// TIA Portal project "Project" (V17)

(* hardware
DEVICE "S71500/ET200MP station_1"  S7-1500 station
   slot 0: "Rail_0"  Rack  6ES7 590-1***0-0AA0
   slot 1: "PLC_1"  CPU 1511-1 PN  6ES7 511-1AK00-0AB0  V1.8
      slot 3: "CPU display_1"  6ES7591-1AA00-0AA0
DEVICE "PC-System_1"  SIMATIC PC station
   slot 0: "SIMATIC PC station"  Rail  SIMATIC PC-Station  V1.0
      slot 125: "Stationmanager"  Station_Manager  V6.0.4
   slot 1: "HMI_RT_1"  WinCC RT Professional  6AV2 105-0xxxx-xxxx  17.0.0.0
   slot 2: "IE general_1"  IE General  IE_CP  V8.2.0
      slot 1: "PROFINET interface"  IEGeneral.Interface.8.2.0
*)

// ===== PLC "PLC_1"  CPU 1511-1 PN =====

VAR_GLOBAL   // PLC tag table "Default tag table"
   "Brake_Out" AT %M0.0 : Bool;
   "Baffle_Out" AT %MW18 : Int;
   "RPM_In" AT %MW2 : Int;
   "OilTemp_In" AT %MW4 : Int;
   "Baffle_En" AT %M0.1 : Bool;
   "Current_In" AT %MW6 : Int;
   "OilPumpVFDsp_Out" AT %MW8 : Int;
   "OilPumpVFDen_Out" AT %M0.2 : Bool;
   "OilFlow_In" AT %MW10 : Int;
   "ProgLang" AT %MW12 : Int;
   "ONS1" AT %M0.3 : Bool;
   "PB_LAD" AT %M0.4 : Bool;
   "PB_FBD" AT %M0.5 : Bool;
   "PB_SCL" AT %M0.6 : Bool;
   "PB_STL" AT %M0.7 : Bool;
   "ONS" AT %M1.0 : Bool;
   "ONS2" AT %M1.1 : Bool;
   "ONS3" AT %M1.2 : Bool;
   "AlarmHorn_Out" AT %M1.3 : Bool;
   "StationInterlock_Out" AT %M1.4 : Bool;
   "OilPumpVFDpct" AT %MW14 : Int;
   "Bafflepct" AT %MW16 : Int;
   "OilTemp" AT %MW20 : Int;
   "OilFlow" AT %MW22 : Int;
   "RPM" AT %MW24 : Int;
   "Current" AT %MW26 : Int;
   "OilPumpVFDOff_PB" AT %M1.5 : Bool;
   "OilPumpVFDHand_PB" AT %M1.6 : Bool;
   "OilPumpVFDAuto_PB" AT %M1.7 : Bool;
   "OilPumpVFDHoa" AT %MW28 : Int;
   "BrakeOff_PB" AT %M2.0 : Bool;
   "BrakeHand_PB" AT %M2.1 : Bool;
   "BrakeAuto_PB" AT %M2.2 : Bool;
   "BrakeHoa" AT %MW30 : Int;
   "AlarmHornOff_PB" AT %M2.3 : Bool;
   "AlarmHornHand_PB" AT %M2.4 : Bool;
   "AlarmHornAuto_PB" AT %M2.5 : Bool;
   "AlarmHornHoa" AT %MW32 : Int;
   "StationInterlockOff_PB" AT %M2.6 : Bool;
   "StationInterlockHand_PB" AT %M2.7 : Bool;
   "StationInterlockAuto_PB" AT %M3.0 : Bool;
   "StationInterlockHoa" AT %MW34 : Int;
   "OilPumpVFD_Ctrl" AT %M3.1 : Bool;
   "Brake_Ctrl" AT %M3.2 : Bool;
   "AlarmHorn_Ctrl" AT %M3.3 : Bool;
   "StationInterlock_Ctrl" AT %M3.4 : Bool;
END_VAR

DATA_BLOCK "SimLogic_DB"   // DB1
{ S7_Optimized_Access := 'TRUE' }
VERSION : 0.1
// stored: InstanceOfName SimLogic
"SimLogic"
BEGIN
END_DATA_BLOCK

DATA_BLOCK "IO_LAD_DB"   // DB2
{ S7_Optimized_Access := 'TRUE' }
VERSION : 0.1
// stored: InstanceOfName IO_LAD
"IO_LAD"
BEGIN
END_DATA_BLOCK

DATA_BLOCK "IO_STL_DB"   // DB4
{ S7_Optimized_Access := 'TRUE' }
VERSION : 0.1
// stored: InstanceOfName IO_STL
"IO_STL"
BEGIN
END_DATA_BLOCK

DATA_BLOCK "IO_SCL_DB"   // DB5
{ S7_Optimized_Access := 'TRUE' }
VERSION : 0.1
// stored: InstanceOfName IO_SCL
"IO_SCL"
BEGIN
END_DATA_BLOCK

DATA_BLOCK "IO_FBD_DB"   // DB6
{ S7_Optimized_Access := 'TRUE' }
VERSION : 0.1
// stored: InstanceOfName IO_FBD
"IO_FBD"
BEGIN
END_DATA_BLOCK

DATA_BLOCK "ALARMS_LAD_DB"   // DB7
{ S7_Optimized_Access := 'TRUE' }
VERSION : 0.1
// stored: InstanceOfName ALARMS_LAD
"ALARMS_LAD"
BEGIN
END_DATA_BLOCK

DATA_BLOCK "HOA_LAD_DB"   // DB8
{ S7_Optimized_Access := 'TRUE' }
VERSION : 0.1
// stored: InstanceOfName HOA_LAD
"HOA_LAD"
BEGIN
END_DATA_BLOCK

DATA_BLOCK "HOA_FBD_DB"   // DB9
{ S7_Optimized_Access := 'TRUE' }
VERSION : 0.1
// stored: InstanceOfName HOA_FBD
"HOA_FBD"
BEGIN
END_DATA_BLOCK

DATA_BLOCK "HOA_SCL_DB"   // DB10
{ S7_Optimized_Access := 'TRUE' }
VERSION : 0.1
// stored: InstanceOfName HOA_SCL
"HOA_SCL"
BEGIN
END_DATA_BLOCK

DATA_BLOCK "HOA_STL_DB"   // DB11
{ S7_Optimized_Access := 'TRUE' }
VERSION : 0.1
// stored: InstanceOfName HOA_STL
"HOA_STL"
BEGIN
END_DATA_BLOCK

// folder: System blocks/Program resources

DATA_BLOCK "IEC_Timer_0_DB_25"   // DB3
{ S7_Optimized_Access := 'TRUE' }
AUTHOR : Simatic
FAMILY : IEC
NAME : IEC_TMR
VERSION : 1.0
// stored: InstanceOfName IEC_TIMER
"IEC_TIMER"
BEGIN
END_DATA_BLOCK

DATA_BLOCK "IEC_Timer_0_DB"   // DB17
{ S7_Optimized_Access := 'TRUE' }
AUTHOR : Simatic
FAMILY : IEC
NAME : IEC_TMR
VERSION : 1.0
// stored: InstanceOfName IEC_TIMER
"IEC_TIMER"
BEGIN
END_DATA_BLOCK

DATA_BLOCK "IEC_Timer_1_DB"   // DB43
{ S7_Optimized_Access := 'TRUE' }
AUTHOR : Simatic
FAMILY : IEC
NAME : IEC_TMR
VERSION : 1.0
// stored: InstanceOfName IEC_TIMER
"IEC_TIMER"
BEGIN
END_DATA_BLOCK

// folder: (top level)

FUNCTION_BLOCK "SimLogic"   // FB1, FBD
{ S7_Optimized_Access := 'TRUE' }
VERSION : 0.1
   VAR
      "TO" : Bool;
      rpmv : Int;
      addrpmv : Bool;
      otsp : Int;
      ott : Int;
      TO1 : Bool;
      TO2 : Bool;
      be2 : Int;
      be3 : Int;
      be1 : Int;
      TO3 : Bool;
   END_VAR
   VAR_TEMP
      bf : Int;
      rpmvt : Int;
      bfr : Real;
   END_VAR
BEGIN

REGION Network 1
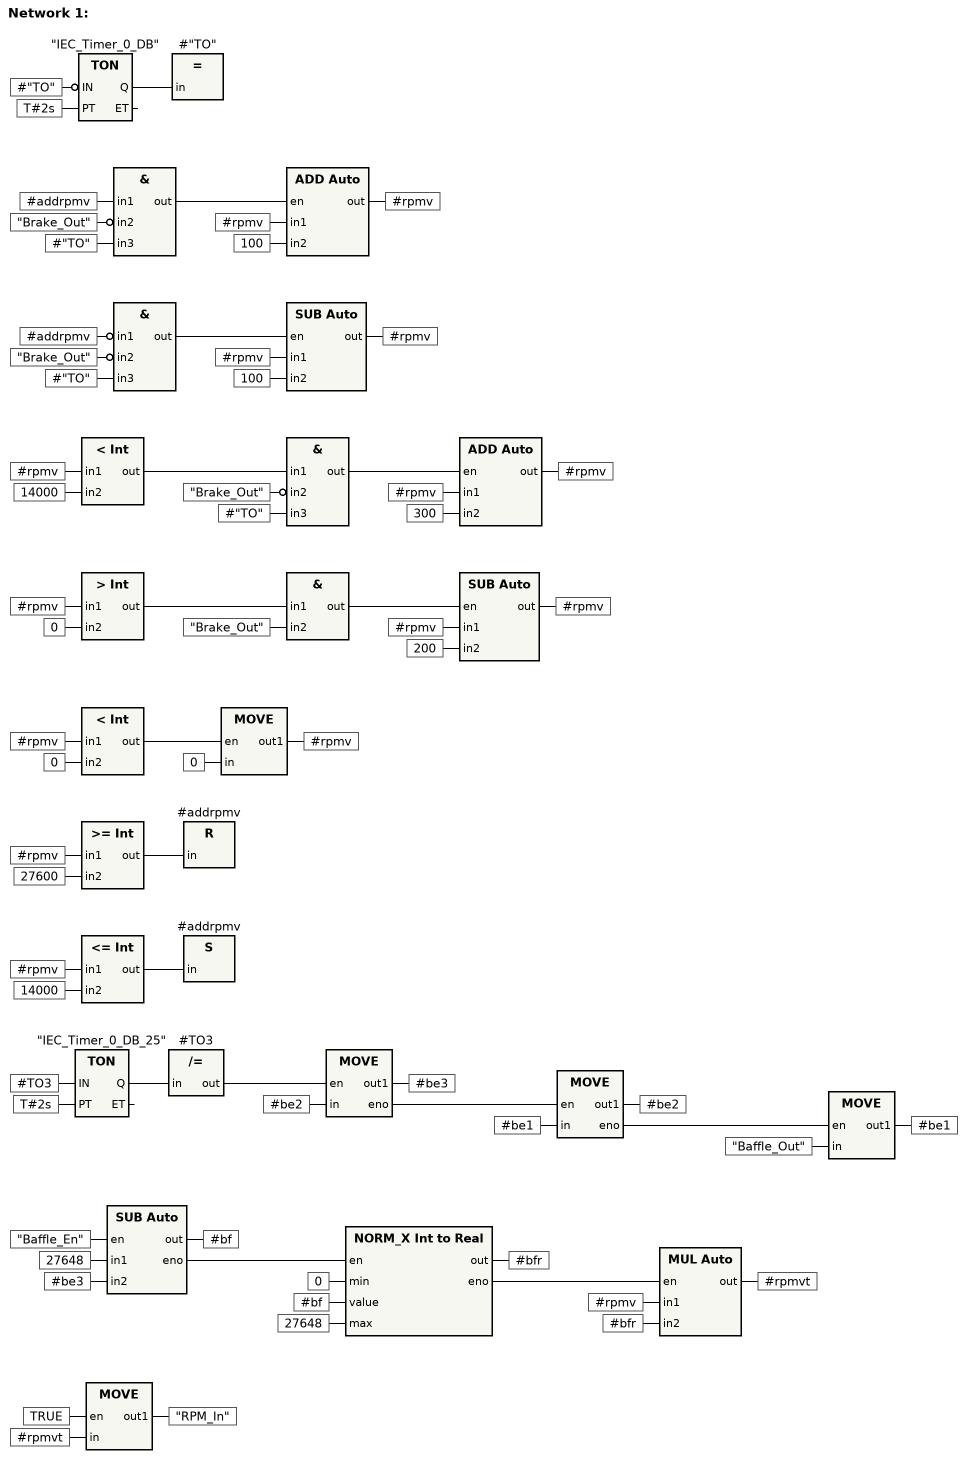
   "IEC_Timer_0_DB".TON(IN := NOT #"TO", PT := T#2s);
   #"TO" := "IEC_Timer_0_DB".Q;
   IF #addrpmv AND NOT "Brake_Out" AND #"TO" THEN #rpmv := #rpmv + 100; END_IF;
   IF NOT #addrpmv AND NOT "Brake_Out" AND #"TO" THEN #rpmv := #rpmv - 100; END_IF;
   IF (#rpmv < 14000) AND NOT "Brake_Out" AND #"TO" THEN #rpmv := #rpmv + 300; END_IF;
   IF (#rpmv > 0) AND "Brake_Out" THEN #rpmv := #rpmv - 200; END_IF;
   IF #rpmv < 0 THEN #rpmv := 0; END_IF;
   IF #rpmv >= 27600 THEN #addrpmv := FALSE; END_IF;
   IF #rpmv <= 14000 THEN #addrpmv := TRUE; END_IF;
   "IEC_Timer_0_DB_25".TON(IN := #TO3, PT := T#2s);
   #TO3 := NOT "IEC_Timer_0_DB_25".Q;
   IF "IEC_Timer_0_DB_25".Q THEN
       #be3 := #be2;
       #be2 := #be1;
       #be1 := "Baffle_Out";
   END_IF;
   IF "Baffle_En" THEN
       #bf := 27648 - #be3;
       #bfr := NORM_X(MIN := 0, VALUE := #bf, MAX := 27648);
       #rpmvt := #rpmv * #bfr;
   END_IF;
   IF TRUE THEN "RPM_In" := #rpmvt; END_IF;
END_REGION

REGION Network 2
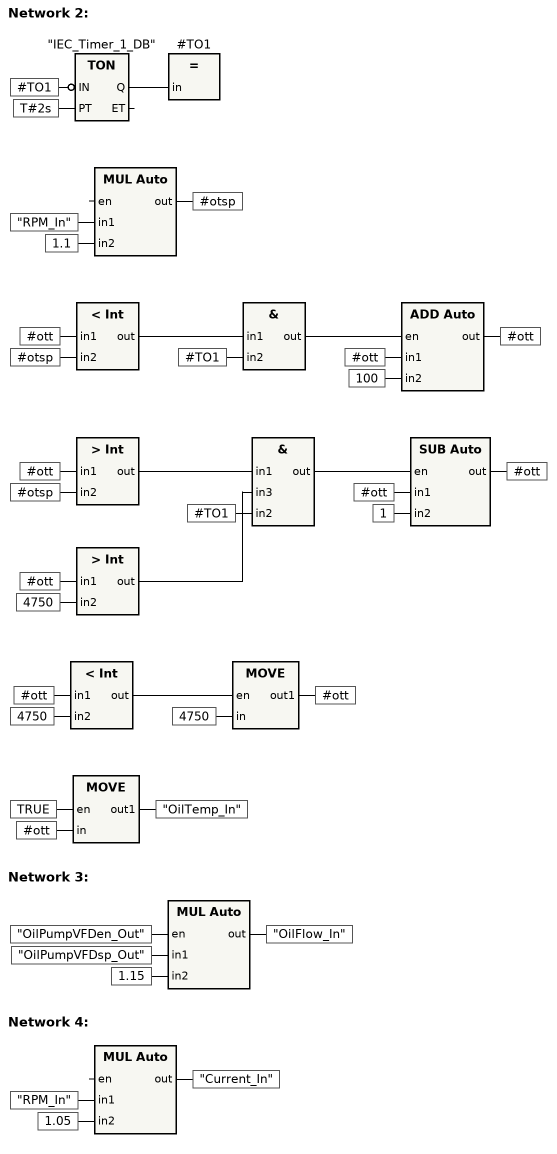
   "IEC_Timer_1_DB".TON(IN := NOT #TO1, PT := T#2s);
   #TO1 := "IEC_Timer_1_DB".Q;
   #otsp := "RPM_In" * 1.1;
   IF (#ott < #otsp) AND #TO1 THEN #ott := #ott + 100; END_IF;
   IF (#ott > #otsp) AND (#ott > 4750) AND #TO1 THEN #ott := #ott - 1; END_IF;
   IF #ott < 4750 THEN #ott := 4750; END_IF;
   IF TRUE THEN "OilTemp_In" := #ott; END_IF;
END_REGION

REGION Network 3
   IF "OilPumpVFDen_Out" THEN "OilFlow_In" := "OilPumpVFDsp_Out" * 1.15; END_IF;
END_REGION

REGION Network 4
   "Current_In" := "RPM_In" * 1.05;
END_REGION
END_FUNCTION_BLOCK

FUNCTION_BLOCK "IO_LAD"   // FB2, LAD
{ S7_Optimized_Access := 'TRUE' }
VERSION : 0.1
BEGIN

REGION Network 1: Digital Outputs
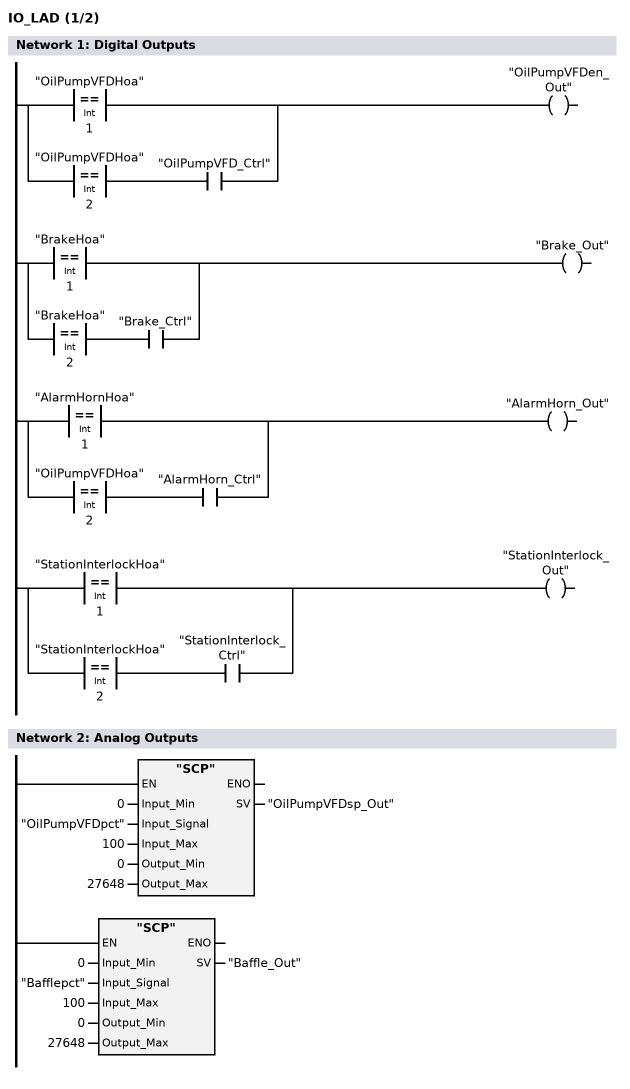
   RUNG wire#powerrail
      { S7_Templates := "SrcType := Int" } EQ_Contact(in1 := "OilPumpVFDHoa", in2 := 1)
      wire#w1
      Coil( "OilPumpVFDen_Out" )
   END_RUNG
   RUNG wire#powerrail
      { S7_Templates := "SrcType := Int" } EQ_Contact(in1 := "OilPumpVFDHoa", in2 := 2)
      Contact( "OilPumpVFD_Ctrl" )
   END_RUNG wire#w1
   RUNG wire#powerrail
      { S7_Templates := "SrcType := Int" } EQ_Contact(in1 := "BrakeHoa", in2 := 1)
      wire#w2
      Coil( "Brake_Out" )
   END_RUNG
   RUNG wire#powerrail
      { S7_Templates := "SrcType := Int" } EQ_Contact(in1 := "BrakeHoa", in2 := 2)
      Contact( "Brake_Ctrl" )
   END_RUNG wire#w2
   RUNG wire#powerrail
      { S7_Templates := "SrcType := Int" } EQ_Contact(in1 := "AlarmHornHoa", in2 := 1)
      wire#w3
      Coil( "AlarmHorn_Out" )
   END_RUNG
   RUNG wire#powerrail
      { S7_Templates := "SrcType := Int" } EQ_Contact(in1 := "OilPumpVFDHoa", in2 := 2)
      Contact( "AlarmHorn_Ctrl" )
   END_RUNG wire#w3
   RUNG wire#powerrail
      { S7_Templates := "SrcType := Int" } EQ_Contact(in1 := "StationInterlockHoa", in2 := 1)
      wire#w4
      Coil( "StationInterlock_Out" )
   END_RUNG
   RUNG wire#powerrail
      { S7_Templates := "SrcType := Int" } EQ_Contact(in1 := "StationInterlockHoa", in2 := 2)
      Contact( "StationInterlock_Ctrl" )
   END_RUNG wire#w4
   // the same network as SCL:
   "OilPumpVFDen_Out" := ("OilPumpVFDHoa" = 1) OR (("OilPumpVFDHoa" = 2) AND "OilPumpVFD_Ctrl");
   "Brake_Out" := ("BrakeHoa" = 1) OR (("BrakeHoa" = 2) AND "Brake_Ctrl");
   "AlarmHorn_Out" := ("AlarmHornHoa" = 1) OR (("OilPumpVFDHoa" = 2) AND "AlarmHorn_Ctrl");
   "StationInterlock_Out" := ("StationInterlockHoa" = 1) OR (("StationInterlockHoa" = 2) AND "StationInterlock_Ctrl");
END_REGION

REGION Network 2: Analog Outputs
   RUNG wire#powerrail
      "SCP"(Input_Min := 0, Input_Signal := "OilPumpVFDpct", Input_Max := 100, Output_Min := 0, Output_Max := 27648, SV => "OilPumpVFDsp_Out")
   END_RUNG
   RUNG wire#powerrail
      "SCP"(Input_Min := 0, Input_Signal := "Bafflepct", Input_Max := 100, Output_Min := 0, Output_Max := 27648, SV => "Baffle_Out")
   END_RUNG
   // the same network as SCL:
   "SCP"(Input_Min := 0,
         Input_Signal := "OilPumpVFDpct",
         Input_Max := 100,
         Output_Min := 0,
         Output_Max := 27648,
         SV => "OilPumpVFDsp_Out");
   "SCP"(Input_Min := 0,
         Input_Signal := "Bafflepct",
         Input_Max := 100,
         Output_Min := 0,
         Output_Max := 27648,
         SV => "Baffle_Out");
END_REGION

REGION Network 3: Analog Inputs
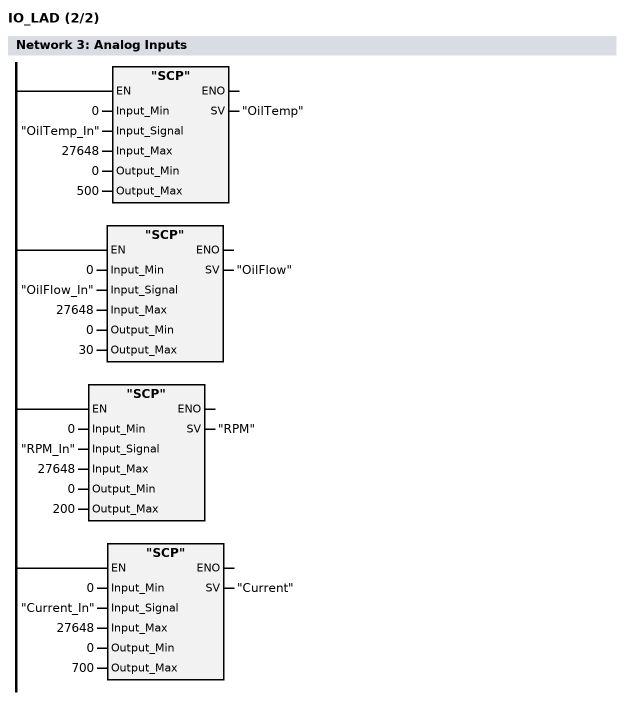
   RUNG wire#powerrail
      "SCP"(Input_Min := 0, Input_Signal := "OilTemp_In", Input_Max := 27648, Output_Min := 0, Output_Max := 500, SV => "OilTemp")
   END_RUNG
   RUNG wire#powerrail
      "SCP"(Input_Min := 0, Input_Signal := "OilFlow_In", Input_Max := 27648, Output_Min := 0, Output_Max := 30, SV => "OilFlow")
   END_RUNG
   RUNG wire#powerrail
      "SCP"(Input_Min := 0, Input_Signal := "RPM_In", Input_Max := 27648, Output_Min := 0, Output_Max := 200, SV => "RPM")
   END_RUNG
   RUNG wire#powerrail
      "SCP"(Input_Min := 0, Input_Signal := "Current_In", Input_Max := 27648, Output_Min := 0, Output_Max := 700, SV => "Current")
   END_RUNG
   // the same network as SCL:
   "SCP"(Input_Min := 0,
         Input_Signal := "OilTemp_In",
         Input_Max := 27648,
         Output_Min := 0,
         Output_Max := 500,
         SV => "OilTemp");
   "SCP"(Input_Min := 0,
         Input_Signal := "OilFlow_In",
         Input_Max := 27648,
         Output_Min := 0,
         Output_Max := 30,
         SV => "OilFlow");
   "SCP"(Input_Min := 0,
         Input_Signal := "RPM_In",
         Input_Max := 27648,
         Output_Min := 0,
         Output_Max := 200,
         SV => "RPM");
   "SCP"(Input_Min := 0,
         Input_Signal := "Current_In",
         Input_Max := 27648,
         Output_Min := 0,
         Output_Max := 700,
         SV => "Current");
END_REGION
END_FUNCTION_BLOCK

FUNCTION_BLOCK "IO_FBD"   // FB3, FBD
{ S7_Optimized_Access := 'TRUE' }
VERSION : 0.1
BEGIN

REGION Network 1: Digital Outputs
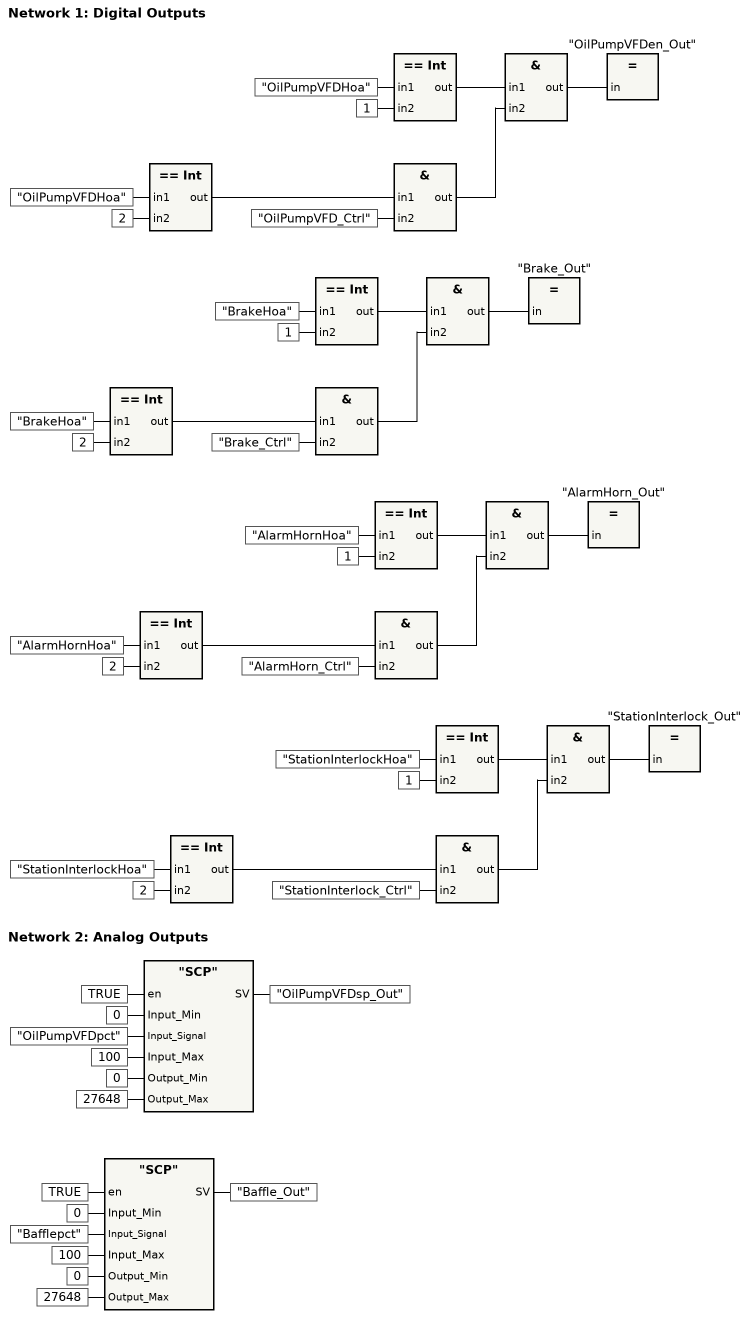
   "OilPumpVFDen_Out" := ("OilPumpVFDHoa" = 1) AND ("OilPumpVFDHoa" = 2) AND "OilPumpVFD_Ctrl";
   "Brake_Out" := ("BrakeHoa" = 1) AND ("BrakeHoa" = 2) AND "Brake_Ctrl";
   "AlarmHorn_Out" := ("AlarmHornHoa" = 1) AND ("AlarmHornHoa" = 2) AND "AlarmHorn_Ctrl";
   "StationInterlock_Out" := ("StationInterlockHoa" = 1) AND ("StationInterlockHoa" = 2) AND "StationInterlock_Ctrl";
END_REGION

REGION Network 2: Analog Outputs
   IF TRUE THEN
       "SCP"(Input_Min := 0,
             Input_Signal := "OilPumpVFDpct",
             Input_Max := 100,
             Output_Min := 0,
             Output_Max := 27648,
             SV => "OilPumpVFDsp_Out");
       "SCP"(Input_Min := 0,
             Input_Signal := "Bafflepct",
             Input_Max := 100,
             Output_Min := 0,
             Output_Max := 27648,
             SV => "Baffle_Out");
   END_IF;
END_REGION

REGION Network 3: Analog Inputs
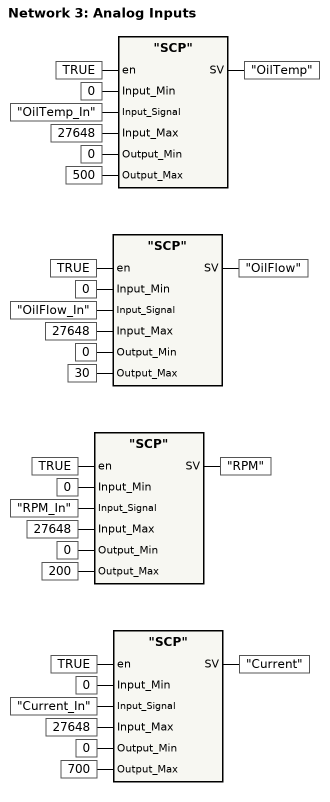
   IF TRUE THEN
       "SCP"(Input_Min := 0,
             Input_Signal := "OilTemp_In",
             Input_Max := 27648,
             Output_Min := 0,
             Output_Max := 500,
             SV => "OilTemp");
       "SCP"(Input_Min := 0,
             Input_Signal := "OilFlow_In",
             Input_Max := 27648,
             Output_Min := 0,
             Output_Max := 30,
             SV => "OilFlow");
       "SCP"(Input_Min := 0,
             Input_Signal := "RPM_In",
             Input_Max := 27648,
             Output_Min := 0,
             Output_Max := 200,
             SV => "RPM");
       "SCP"(Input_Min := 0,
             Input_Signal := "Current_In",
             Input_Max := 27648,
             Output_Min := 0,
             Output_Max := 700,
             SV => "Current");
   END_IF;
END_REGION
END_FUNCTION_BLOCK

FUNCTION_BLOCK "IO_SCL"   // FB4, SCL
{ S7_Optimized_Access := 'TRUE' }
VERSION : 0.1
BEGIN
   //Digital Ouputs
   IF "OilPumpVFDHoa" = 0 OR ("OilPumpVFDHoa" = 2 AND NOT "OilPumpVFD_Ctrl") THEN
       "OilPumpVFDen_Out" := 0;
   END_IF;

   IF "OilPumpVFDHoa" = 1 OR ("OilPumpVFDHoa" = 2 AND "OilPumpVFD_Ctrl") THEN
       "OilPumpVFDen_Out" := 1;
   END_IF;


   IF "BrakeHoa" = 0 OR ("BrakeHoa" = 2 AND NOT "Brake_Ctrl") THEN
       "Brake_Out" := 0;
   END_IF;

   IF "BrakeHoa" = 1 OR ("BrakeHoa" = 2 AND "Brake_Ctrl") THEN
       "Brake_Out" := 1;
   END_IF;


   IF "AlarmHornHoa" = 0 OR ("AlarmHornHoa" = 2 AND NOT "AlarmHorn_Ctrl") THEN
       "AlarmHorn_Out" := 0;
   END_IF;

   IF "AlarmHornHoa" = 1 OR ("AlarmHornHoa" = 2 AND "AlarmHorn_Ctrl") THEN
       "AlarmHorn_Out" := 1;
   END_IF;


   IF "StationInterlockHoa" = 0 OR ("StationInterlockHoa" = 2 AND NOT "StationInterlock_Ctrl") THEN
       "StationInterlock_Out" := 0;
   END_IF;

   IF "StationInterlockHoa" = 1 OR ("StationInterlockHoa" = 2 AND "StationInterlock_Ctrl") THEN
       "StationInterlock_Out" := 1;
   END_IF;

   // Analog Outputs
   "SCP"(Input_Min:=0,
         Input_Signal:="OilPumpVFDpct",
         Input_Max:=100,
         Output_Min:=0,
         Output_Max:=27648,
         SV=>"OilPumpVFDsp_Out");

   "SCP"(Input_Min := 0,
         Input_Signal := "Bafflepct",
         Input_Max := 100,
         Output_Min := 0,
         Output_Max := 27648,
         SV => "Baffle_Out");

   //Analog Inputs
   "SCP"(Input_Min := 0,
         Input_Signal := "OilTemp_In",
         Input_Max := 27648,
         Output_Min := 0,
         Output_Max := 500,
         SV => "OilTemp");

   "SCP"(Input_Min := 0,
         Input_Signal := "OilFlow_In",
         Input_Max := 27648,
         Output_Min := 0,
         Output_Max := 30,
         SV => "OilFlow");

   "SCP"(Input_Min := 0,
         Input_Signal := "RPM_In",
         Input_Max := 27648,
         Output_Min := 0,
         Output_Max := 200,
         SV => "RPM");

   "SCP"(Input_Min := 0,
         Input_Signal := "Current_In",
         Input_Max := 27648,
         Output_Min := 0,
         Output_Max := 700,
         SV => "Current");
END_FUNCTION_BLOCK

FUNCTION_BLOCK "IO_STL"   // FB5, STL
{ S7_Optimized_Access := 'TRUE' }
VERSION : 0.1
BEGIN

REGION Network 1
   //Digital Ouputs
   OilPumpVFD:L     "OilPumpVFDHoa";
         L     0;
         ==I;
         JC    ResetOilPumpVFD;
         CLR;
         L     "OilPumpVFDHoa";
         L     1;
         ==I;
         JC    SetOilPumpVFD;
         CLR;
         L     "OilPumpVFDHoa";
         L     2;
         ==I;
         JC    AutoOilPumpVFD;

   AutoOilPumpVFD:A     "OilPumpVFD_Ctrl";
         JC    SetOilPumpVFD;
         JU    Brake;
   SetOilPumpVFD:S     "OilPumpVFDen_Out";
         JU    Brake;
   ResetOilPumpVFD:R     "OilPumpVFDen_Out";
         JU    Brake;


   Brake:L     "BrakeHoa";
         L     0;
         ==I;
         JC    ResetBrake;
         CLR;
         L     "BrakeHoa";
         L     1;
         ==I;
         JC    SetBrake;
         CLR;
         L     "BrakeHoa";
         L     2;
         ==I;
         JC    AutoBrake;

   AutoBrake:A     "Brake_Ctrl";
         JC    SetBrake;
         JU    AlarmHorn;
   SetBrake:S     "Brake_Out";
         JU    AlarmHorn;
   ResetBrake:R     "Brake_Out";
         JU    AlarmHorn;

   AlarmHorn:L     "AlarmHornHoa";
         L     0;
         ==I;
         JC    ResetAlarmHorn;
         CLR;
         L     "AlarmHornHoa";
         L     1;
         ==I;
         JC    SetAlarmHorn;
         CLR;
         L     "AlarmHornHoa";
         L     2;
         ==I;
         JC    AutoAlarmHorn;

   AutoAlarmHorn:A     "AlarmHorn_Ctrl";
         JC    SetAlarmHorn;
         JU    StationInterlock;
   SetAlarmHorn:S     "AlarmHorn_Out";
         JU    StationInterlock;
   ResetAlarmHorn:R     "AlarmHorn_Out";
         JU    StationInterlock;

   StationInterlock:L     "StationInterlockHoa";
         L     0;
         ==I;
         JC    ResetStationInterlock;
         CLR;
         L     "StationInterlockHoa";
         L     1;
         ==I;
         JC    SetStationInterlock;
         CLR;
         L     "StationInterlockHoa";
         L     2;
         ==I;
         JC    AutoStationInterlock;

   AutoStationInterlock:A     "StationInterlock_Ctrl";
         JC    SetStationInterlock;
         JU    AnalogOutputs;
   SetStationInterlock:S     "StationInterlock_Out";
         JU    AnalogOutputs;
   ResetStationInterlock:R     "StationInterlock_Out";
         JU    AnalogOutputs;


   //Analog Outputs
   AnalogOutputs:CALL  "SCP"
         ( Input_Min    := 0,
           Input_Signal := "OilPumpVFDpct",
           Input_Max    := 100,
           Output_Min   := 0,
           Output_Max   := 27648,
           SV           := "OilPumpVFDsp_Out"
         );

         CALL  "SCP"
         ( Input_Min    := 0,
           Input_Signal := "Bafflepct",
           Input_Max    := 100,
           Output_Min   := 0,
           Output_Max   := 27648,
           SV           := "Baffle_Out"
         );

   //Analog Inputs
   AnalogInputs:CALL  "SCP"
         ( Input_Min    := 0,
           Input_Signal := "OilTemp_In",
           Input_Max    := 27648,
           Output_Min   := 0,
           Output_Max   := 500,
           SV           := "OilTemp"
         );

         CALL  "SCP"
         ( Input_Min    := 0,
           Input_Signal := "OilFlow_In",
           Input_Max    := 27648,
           Output_Min   := 0,
           Output_Max   := 30,
           SV           := "OilFlow"
         );

         CALL  "SCP"
         ( Input_Min    := 0,
           Input_Signal := "RPM_In",
           Input_Max    := 27648,
           Output_Min   := 0,
           Output_Max   := 200,
           SV           := "RPM"
         );

         CALL  "SCP"
         ( Input_Min    := 0,
           Input_Signal := "Current_In",
           Input_Max    := 27648,
           Output_Min   := 0,
           Output_Max   := 700,
           SV           := "Current"
         );
END_REGION
END_FUNCTION_BLOCK

FUNCTION_BLOCK "ALARMS_LAD"   // FB6, LAD
{ S7_Optimized_Access := 'TRUE' }
VERSION : 0.1
BEGIN
END_FUNCTION_BLOCK

FUNCTION_BLOCK "HOA_LAD"   // FB7, LAD
{ S7_Optimized_Access := 'TRUE' }
VERSION : 0.1
   VAR
      OS1 : Bool;
      OS2 : Bool;
      OS3 : Bool;
      OS4 : Bool;
      OS5 : Bool;
      OS6 : Bool;
      OS7 : Bool;
      OS8 : Bool;
      OS9 : Bool;
      OS10 : Bool;
      OS11 : Bool;
      OS12 : Bool;
   END_VAR
   VAR_TEMP   // added for the SCL form of the ladder/FBD networks
      _w1 : Bool;
      _w2 : Bool;
      _w3 : Bool;
   END_VAR
BEGIN

REGION Network 1: OilPumpVFD
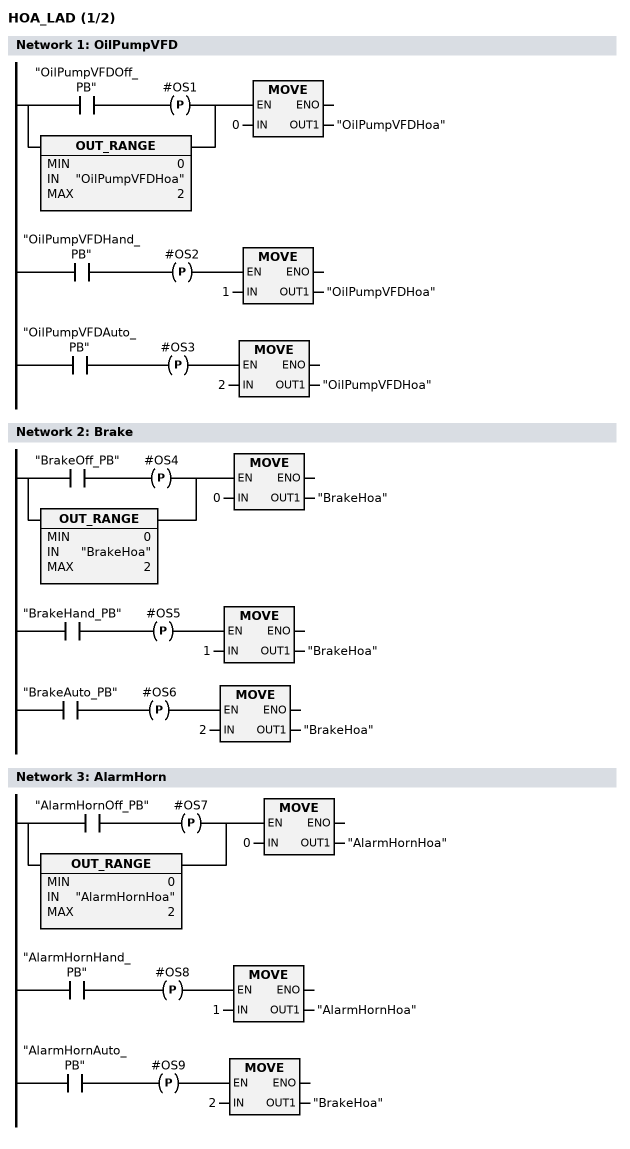
   #_w1 := "OilPumpVFDOff_PB" AND NOT #OS1;   // rising edge
   #OS1 := "OilPumpVFDOff_PB";
   IF #_w1 OR ("OilPumpVFDHoa" < 0) OR ("OilPumpVFDHoa" > 2) THEN "OilPumpVFDHoa" := 0; END_IF;
   #_w2 := "OilPumpVFDHand_PB" AND NOT #OS2;   // rising edge
   #OS2 := "OilPumpVFDHand_PB";
   IF #_w2 THEN "OilPumpVFDHoa" := 1; END_IF;
   #_w3 := "OilPumpVFDAuto_PB" AND NOT #OS3;   // rising edge
   #OS3 := "OilPumpVFDAuto_PB";
   IF #_w3 THEN "OilPumpVFDHoa" := 2; END_IF;
END_REGION

REGION Network 2: Brake
   #_w1 := "BrakeOff_PB" AND NOT #OS4;   // rising edge
   #OS4 := "BrakeOff_PB";
   IF #_w1 OR ("BrakeHoa" < 0) OR ("BrakeHoa" > 2) THEN "BrakeHoa" := 0; END_IF;
   #_w2 := "BrakeHand_PB" AND NOT #OS5;   // rising edge
   #OS5 := "BrakeHand_PB";
   IF #_w2 THEN "BrakeHoa" := 1; END_IF;
   #_w3 := "BrakeAuto_PB" AND NOT #OS6;   // rising edge
   #OS6 := "BrakeAuto_PB";
   IF #_w3 THEN "BrakeHoa" := 2; END_IF;
END_REGION

REGION Network 3: AlarmHorn
   #_w1 := "AlarmHornOff_PB" AND NOT #OS7;   // rising edge
   #OS7 := "AlarmHornOff_PB";
   IF #_w1 OR ("AlarmHornHoa" < 0) OR ("AlarmHornHoa" > 2) THEN "AlarmHornHoa" := 0; END_IF;
   #_w2 := "AlarmHornHand_PB" AND NOT #OS8;   // rising edge
   #OS8 := "AlarmHornHand_PB";
   IF #_w2 THEN "AlarmHornHoa" := 1; END_IF;
   #_w3 := "AlarmHornAuto_PB" AND NOT #OS9;   // rising edge
   #OS9 := "AlarmHornAuto_PB";
   IF #_w3 THEN "BrakeHoa" := 2; END_IF;
END_REGION

REGION Network 4: StationInterlock
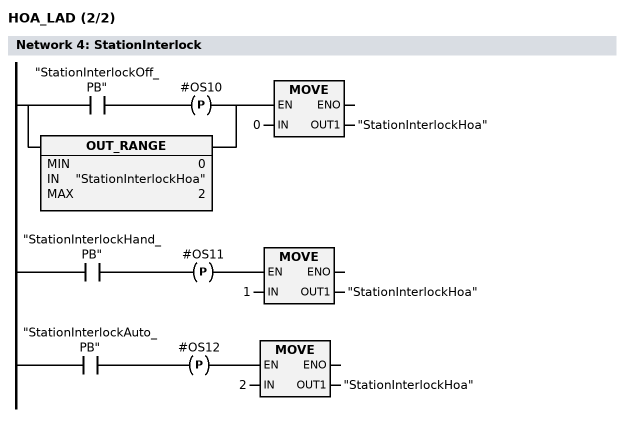
   #_w1 := "StationInterlockOff_PB" AND NOT #OS10;   // rising edge
   #OS10 := "StationInterlockOff_PB";
   IF #_w1 OR ("StationInterlockHoa" < 0) OR ("StationInterlockHoa" > 2) THEN
       "StationInterlockHoa" := 0;
   END_IF;
   #_w2 := "StationInterlockHand_PB" AND NOT #OS11;   // rising edge
   #OS11 := "StationInterlockHand_PB";
   IF #_w2 THEN "StationInterlockHoa" := 1; END_IF;
   #_w3 := "StationInterlockAuto_PB" AND NOT #OS12;   // rising edge
   #OS12 := "StationInterlockAuto_PB";
   IF #_w3 THEN "StationInterlockHoa" := 2; END_IF;
END_REGION
END_FUNCTION_BLOCK

FUNCTION_BLOCK "HOA_FBD"   // FB8, FBD
{ S7_Optimized_Access := 'TRUE' }
VERSION : 0.1
   VAR
      OS1 : Bool;
      OS2 : Bool;
      OS3 : Bool;
      OS4 : Bool;
      OS5 : Bool;
      OS6 : Bool;
      OS7 : Bool;
      OS8 : Bool;
      OS9 : Bool;
      OS10 : Bool;
      OS11 : Bool;
      OS12 : Bool;
   END_VAR
   VAR_TEMP   // added for the SCL form of the ladder/FBD networks
      _w1 : Bool;
      _w2 : Bool;
      _w3 : Bool;
   END_VAR
BEGIN

REGION Network 1: OilPumpVFD
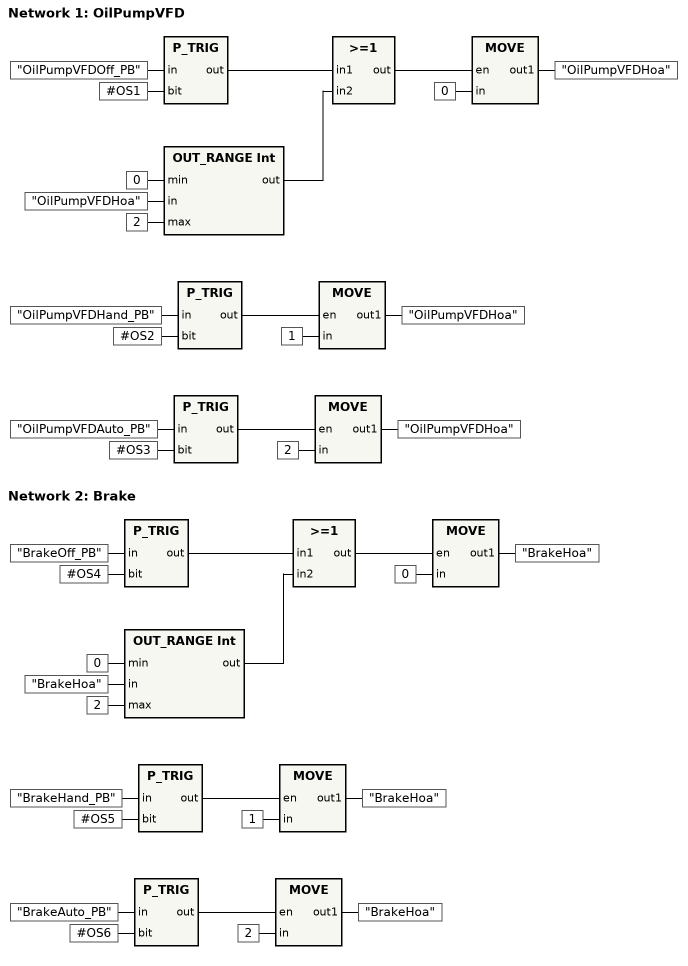
   #_w1 := "OilPumpVFDOff_PB" AND NOT #OS1;   // rising edge
   #OS1 := "OilPumpVFDOff_PB";
   IF #_w1 OR ("OilPumpVFDHoa" < 0) OR ("OilPumpVFDHoa" > 2) THEN "OilPumpVFDHoa" := 0; END_IF;
   #_w2 := "OilPumpVFDHand_PB" AND NOT #OS2;   // rising edge
   #OS2 := "OilPumpVFDHand_PB";
   IF #_w2 THEN "OilPumpVFDHoa" := 1; END_IF;
   #_w3 := "OilPumpVFDAuto_PB" AND NOT #OS3;   // rising edge
   #OS3 := "OilPumpVFDAuto_PB";
   IF #_w3 THEN "OilPumpVFDHoa" := 2; END_IF;
END_REGION

REGION Network 2: Brake
   #_w1 := "BrakeOff_PB" AND NOT #OS4;   // rising edge
   #OS4 := "BrakeOff_PB";
   IF #_w1 OR ("BrakeHoa" < 0) OR ("BrakeHoa" > 2) THEN "BrakeHoa" := 0; END_IF;
   #_w2 := "BrakeHand_PB" AND NOT #OS5;   // rising edge
   #OS5 := "BrakeHand_PB";
   IF #_w2 THEN "BrakeHoa" := 1; END_IF;
   #_w3 := "BrakeAuto_PB" AND NOT #OS6;   // rising edge
   #OS6 := "BrakeAuto_PB";
   IF #_w3 THEN "BrakeHoa" := 2; END_IF;
END_REGION

REGION Network 3: AlarmHorn
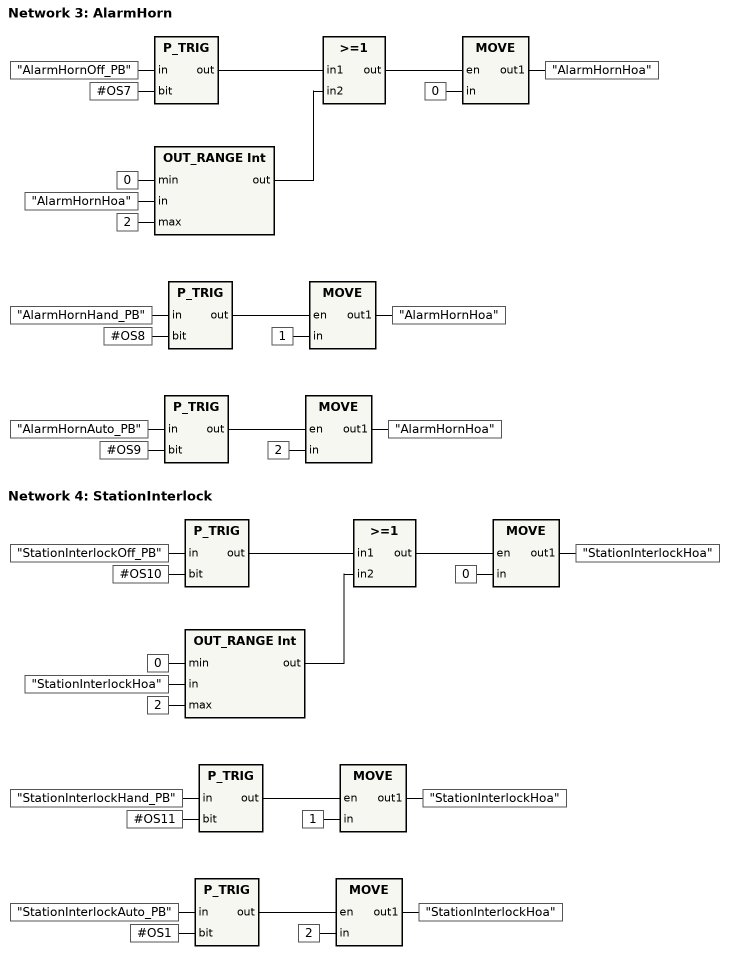
   #_w1 := "AlarmHornOff_PB" AND NOT #OS7;   // rising edge
   #OS7 := "AlarmHornOff_PB";
   IF #_w1 OR ("AlarmHornHoa" < 0) OR ("AlarmHornHoa" > 2) THEN "AlarmHornHoa" := 0; END_IF;
   #_w2 := "AlarmHornHand_PB" AND NOT #OS8;   // rising edge
   #OS8 := "AlarmHornHand_PB";
   IF #_w2 THEN "AlarmHornHoa" := 1; END_IF;
   #_w3 := "AlarmHornAuto_PB" AND NOT #OS9;   // rising edge
   #OS9 := "AlarmHornAuto_PB";
   IF #_w3 THEN "AlarmHornHoa" := 2; END_IF;
END_REGION

REGION Network 4: StationInterlock
   #_w1 := "StationInterlockOff_PB" AND NOT #OS10;   // rising edge
   #OS10 := "StationInterlockOff_PB";
   IF #_w1 OR ("StationInterlockHoa" < 0) OR ("StationInterlockHoa" > 2) THEN
       "StationInterlockHoa" := 0;
   END_IF;
   #_w2 := "StationInterlockHand_PB" AND NOT #OS11;   // rising edge
   #OS11 := "StationInterlockHand_PB";
   IF #_w2 THEN "StationInterlockHoa" := 1; END_IF;
   #_w3 := "StationInterlockAuto_PB" AND NOT #OS1;   // rising edge
   #OS1 := "StationInterlockAuto_PB";
   IF #_w3 THEN "StationInterlockHoa" := 2; END_IF;
END_REGION
END_FUNCTION_BLOCK

FUNCTION_BLOCK "HOA_SCL"   // FB9, SCL
{ S7_Optimized_Access := 'TRUE' }
VERSION : 0.1
BEGIN
   // OilPumpVFD
   IF "OilPumpVFDHoa" < 0 OR "OilPumpVFDHoa" > 2 THEN
       "OilPumpVFDHoa" := 0;
   END_IF;

   IF "OilPumpVFDOff_PB" AND "OilPumpVFDHoa" <> 0 THEN
       "OilPumpVFDHoa" := 0;
   END_IF;

   IF "OilPumpVFDHand_PB" AND "OilPumpVFDHoa" <> 1 THEN
       "OilPumpVFDHoa" := 1;
   END_IF;

   IF "OilPumpVFDAuto_PB" AND "OilPumpVFDHoa" <> 2 THEN
       "OilPumpVFDHoa" := 2;
   END_IF;

   //Brake
   IF "BrakeHoa" < 0 OR "BrakeHoa" > 2 THEN
       "BrakeHoa" := 0;
   END_IF;

   IF "BrakeOff_PB" AND "BrakeHoa" <> 0 THEN
       "BrakeHoa" := 0;
   END_IF;

   IF "BrakeHand_PB" AND "BrakeHoa" <> 1 THEN
       "BrakeHoa" := 1;
   END_IF;

   IF "BrakeAuto_PB" AND "BrakeHoa" <> 2 THEN
       "BrakeHoa" := 2;
   END_IF;

   //AlarmHorn
   IF "AlarmHornHoa" < 0 OR "AlarmHornHoa" > 2 THEN
       "AlarmHornHoa" := 0;
   END_IF;

   IF "AlarmHornOff_PB" AND "AlarmHornHoa" <> 0 THEN
       "AlarmHornHoa" := 0;
   END_IF;

   IF "AlarmHornHand_PB" AND "AlarmHornHoa" <> 1 THEN
       "AlarmHornHoa" := 1;
   END_IF;

   IF "AlarmHornAuto_PB" AND "AlarmHornHoa" <> 2 THEN
       "AlarmHornHoa" := 2;
   END_IF;

   //StationInterlock
   IF "StationInterlockHoa" < 0 OR "StationInterlockHoa" > 2 THEN
       "StationInterlockHoa" := 0;
   END_IF;

   IF "StationInterlockOff_PB" AND "StationInterlockHoa" <> 0 THEN
       "StationInterlockHoa" := 0;
   END_IF;

   IF "StationInterlockHand_PB" AND "StationInterlockHoa" <> 1 THEN
       "StationInterlockHoa" := 1;
   END_IF;

   IF "StationInterlockAuto_PB" AND "StationInterlockHoa" <> 2 THEN
       "StationInterlockHoa" := 2;
   END_IF;
END_FUNCTION_BLOCK

FUNCTION_BLOCK "HOA_STL"   // FB10, STL
{ S7_Optimized_Access := 'TRUE' }
VERSION : 0.1
   VAR
      OS1 : Bool;
      OS2 : Bool;
      OS3 : Bool;
      OS4 : Bool;
      OS5 : Bool;
      OS6 : Bool;
      OS7 : Bool;
      OS8 : Bool;
      OS9 : Bool;
      OS10 : Bool;
      OS11 : Bool;
      OS12 : Bool;
   END_VAR
BEGIN

REGION Network 1
   OilPumpVFD:L     "OilPumpVFDHoa";
         L     0;
         <I;
         JC    SetOilPumpVFDHoaZero;
         CLR;
         L     "OilPumpVFDHoa";
         L     2;
         >I;
         JC    SetOilPumpVFDHoaZero;
         CLR;
         A     "OilPumpVFDOff_PB";
         FP    #OS1;
         JC    SetOilPumpVFDHoaZero;
         CLR;
         A     "OilPumpVFDHand_PB";
         FP    #OS2;
         JC    SetOilPumpVFDHoaOne;
         CLR;
         A     "OilPumpVFDAuto_PB";
         FP    #OS3;
         JC    SetOilPumpVFDHoaTwo;
         JU    EndOfLine;

   SetOilPumpVFDHoaZero:L     0;
         T     "OilPumpVFDHoa";
         BE;

   SetOilPumpVFDHoaOne:L     1;
         T     "OilPumpVFDHoa";
         BE;

   SetOilPumpVFDHoaTwo:L     2;
         T     "OilPumpVFDHoa";
         BE;

   EndOfLine:BE;


   Brake:L     "BrakeHoa";
         L     0;
         <I;
         JC    SetBrakeHoaZero;
         CLR;
         L     "BrakeHoa";
         L     2;
         >I;
         JC    SetBrakeHoaZero;
         CLR;
         A     "BrakeOff_PB";
         FP    #OS4;
         JC    SetBrakeHoaZero;
         CLR;
         A     "BrakeHand_PB";
         FP    #OS5;
         JC    SetBrakeHoaOne;
         CLR;
         A     "BrakeAuto_PB";
         FP    #OS6;
         JC    SetBrakeHoaTwo;
         JU    EndOfLine2;

   SetBrakeHoaZero:L     0;
         T     "BrakeHoa";
         BE;

   SetBrakeHoaOne:L     1;
         T     "BrakeHoa";
         BE;

   SetBrakeHoaTwo:L     2;
         T     "BrakeHoa";
         BE;

   EndOfLine2:BE;

   AlarmHorn:L     "AlarmHornHoa";
         L     0;
         <I;
         JC    SetAlarmHornHoaZero;
         CLR;
         L     "AlarmHornHoa";
         L     2;
         >I;
         JC    SetAlarmHornHoaZero;
         CLR;
         A     "AlarmHornOff_PB";
         FP    #OS7;
         JC    SetAlarmHornHoaZero;
         CLR;
         A     "AlarmHornHand_PB";
         FP    #OS8;
         JC    SetAlarmHornHoaOne;
         CLR;
         A     "AlarmHornAuto_PB";
         FP    #OS9;
         JC    SetAlarmHornHoaTwo;
         JU    EndOfLine3;

   SetAlarmHornHoaZero:L     0;
         T     "AlarmHornHoa";
         BE;

   SetAlarmHornHoaOne:L     1;
         T     "AlarmHornHoa";
         BE;

   SetAlarmHornHoaTwo:L     2;
         T     "AlarmHornHoa";
         BE;

   EndOfLine3:BE;


   StationInterlock:L     "StationInterlockHoa";
         L     0;
         <I;
         JC    SetStationInterlockHoaZero;
         CLR;
         L     "StationInterlockHoa";
         L     2;
         >I;
         JC    SetStationInterlockHoaZero;
         CLR;
         A     "StationInterlockOff_PB";
         FP    #OS10;
         JC    SetStationInterlockHoaZero;
         CLR;
         A     "StationInterlockHand_PB";
         FP    #OS11;
         JC    SetStationInterlockHoaOne;
         CLR;
         A     "StationInterlockAuto_PB";
         FP    #OS12;
         JC    SetStationInterlockHoaTwo;
         JU    EndOfLine4;

   SetStationInterlockHoaZero:L     0;
         T     "StationInterlockHoa";
         BE;

   SetStationInterlockHoaOne:L     1;
         T     "StationInterlockHoa";
         BE;

   SetStationInterlockHoaTwo:L     2;
         T     "StationInterlockHoa";
         BE;

   EndOfLine4:BE;
END_REGION
END_FUNCTION_BLOCK

FUNCTION "SCP" : Void   // FC1, FBD
{ S7_Optimized_Access := 'TRUE' }
VERSION : 0.1
   VAR_INPUT
      Input_Min : Int;
      Input_Signal : Int;
      Input_Max : Int;
      Output_Min : Int;
      Output_Max : Int;
   END_VAR
   VAR_OUTPUT
      SV : Int;
   END_VAR
   VAR_TEMP
      tv : Real;
   END_VAR
BEGIN

REGION Network 1
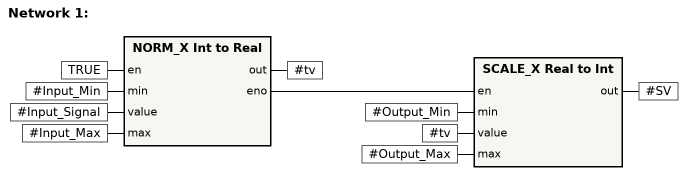
   IF TRUE THEN
       #tv := NORM_X(MIN := #Input_Min, VALUE := #Input_Signal, MAX := #Input_Max);
       #SV := SCALE_X(MIN := #Output_Min, VALUE := #tv, MAX := #Output_Max);
   END_IF;
END_REGION
END_FUNCTION

ORGANIZATION_BLOCK "Main"   // OB1, LAD, ProgramCycle
TITLE = "Main Program Sweep (Cycle)"
{ S7_Optimized_Access := 'TRUE' }
VERSION : 0.1
   VAR_INPUT
      Initial_Call : Bool;   // Initial call of this OB
      Remanence : Bool;   // =True, if remanent data are available
   END_VAR
   VAR_TEMP
      SequenceInit : Bool;
      InitSequence : Bool;
   END_VAR
   VAR_TEMP   // added for the SCL form of the ladder/FBD networks
      _w1 : Bool;
      _w2 : Bool;
      _w3 : Bool;
      _w4 : Bool;
   END_VAR
BEGIN

REGION Network 1
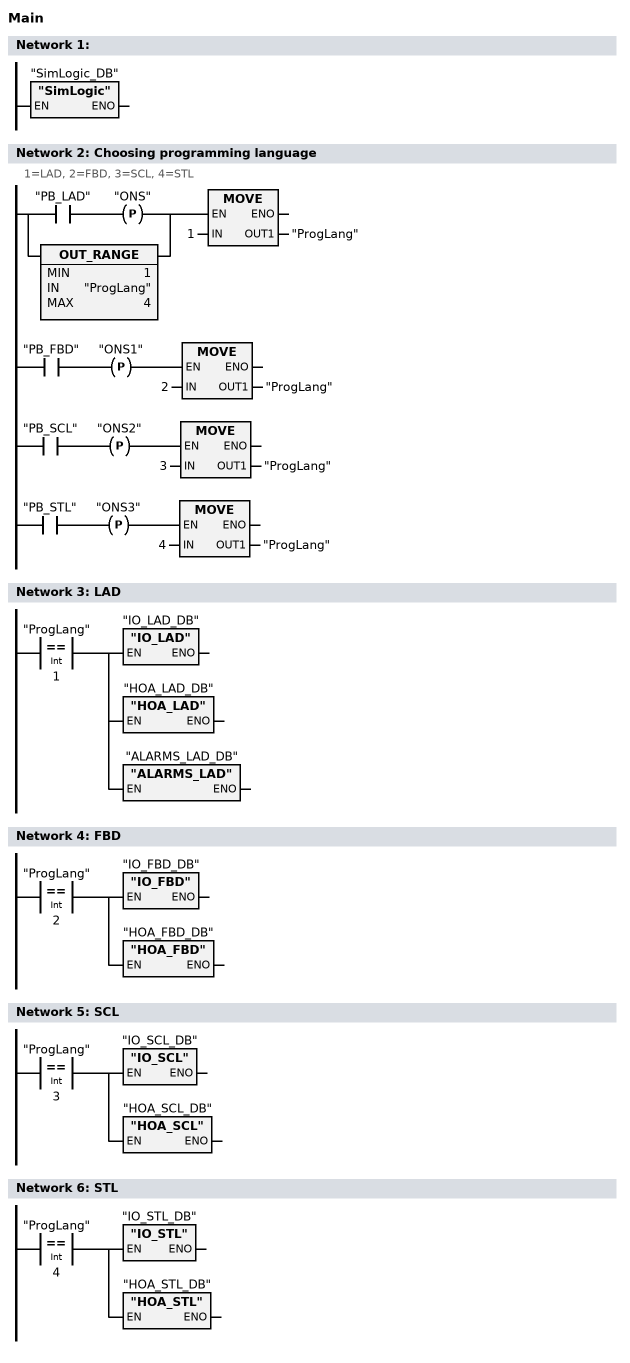
   RUNG wire#powerrail
      "SimLogic_DB"()
   END_RUNG
   // the same network as SCL:
   "SimLogic_DB"();   // "SimLogic"
END_REGION

REGION Network 2: Choosing programming language
   // 1=LAD, 2=FBD, 3=SCL, 4=STL
   #_w1 := "PB_LAD" AND NOT "ONS";   // rising edge
   "ONS" := "PB_LAD";
   IF #_w1 OR ("ProgLang" < 1) OR ("ProgLang" > 4) THEN "ProgLang" := 1; END_IF;
   #_w2 := "PB_FBD" AND NOT "ONS1";   // rising edge
   "ONS1" := "PB_FBD";
   IF #_w2 THEN "ProgLang" := 2; END_IF;
   #_w3 := "PB_SCL" AND NOT "ONS2";   // rising edge
   "ONS2" := "PB_SCL";
   IF #_w3 THEN "ProgLang" := 3; END_IF;
   #_w4 := "PB_STL" AND NOT "ONS3";   // rising edge
   "ONS3" := "PB_STL";
   IF #_w4 THEN "ProgLang" := 4; END_IF;
END_REGION

REGION Network 3: LAD
   RUNG wire#powerrail
      { S7_Templates := "SrcType := Int" } EQ_Contact(in1 := "ProgLang", in2 := 1)
      wire#w1
      "IO_LAD_DB"()
   END_RUNG
   RUNG wire#w1
      "HOA_LAD_DB"()
   END_RUNG
   RUNG wire#w1
      "ALARMS_LAD_DB"()
   END_RUNG
   // the same network as SCL:
   #_w1 := "ProgLang" = 1;
   IF #_w1 THEN
       "IO_LAD_DB"();   // "IO_LAD"
       "HOA_LAD_DB"();   // "HOA_LAD"
       "ALARMS_LAD_DB"();   // "ALARMS_LAD"
   END_IF;
END_REGION

REGION Network 4: FBD
   RUNG wire#powerrail
      { S7_Templates := "SrcType := Int" } EQ_Contact(in1 := "ProgLang", in2 := 2)
      wire#w1
      "IO_FBD_DB"()
   END_RUNG
   RUNG wire#w1
      "HOA_FBD_DB"()
   END_RUNG
   // the same network as SCL:
   #_w1 := "ProgLang" = 2;
   IF #_w1 THEN
       "IO_FBD_DB"();   // "IO_FBD"
       "HOA_FBD_DB"();   // "HOA_FBD"
   END_IF;
END_REGION

REGION Network 5: SCL
   RUNG wire#powerrail
      { S7_Templates := "SrcType := Int" } EQ_Contact(in1 := "ProgLang", in2 := 3)
      wire#w1
      "IO_SCL_DB"()
   END_RUNG
   RUNG wire#w1
      "HOA_SCL_DB"()
   END_RUNG
   // the same network as SCL:
   #_w1 := "ProgLang" = 3;
   IF #_w1 THEN
       "IO_SCL_DB"();   // "IO_SCL"
       "HOA_SCL_DB"();   // "HOA_SCL"
   END_IF;
END_REGION

REGION Network 6: STL
   RUNG wire#powerrail
      { S7_Templates := "SrcType := Int" } EQ_Contact(in1 := "ProgLang", in2 := 4)
      wire#w1
      "IO_STL_DB"()
   END_RUNG
   RUNG wire#w1
      "HOA_STL_DB"()
   END_RUNG
   // the same network as SCL:
   #_w1 := "ProgLang" = 4;
   IF #_w1 THEN
       "IO_STL_DB"();   // "IO_STL"
       "HOA_STL_DB"();   // "HOA_STL"
   END_IF;
END_REGION
END_ORGANIZATION_BLOCK

(* ===== HMI "HMI_RT_1" =====
connection "HMI_Connection_1": S71200_TCP_IP, SCADA_S7_1500_OMS
*)